// SIMATIC S7-200 SMART project (STEP 7-Micro/WIN SMART), CPU SR40

SYMBOL_TABLE 系统符号
Always_On        SM0.0    // 始终接通
First_Scan_On    SM0.1    // 仅在第一个扫描周期时接通
END_SYMBOL_TABLE

ORGANIZATION_BLOCK MAIN:OB1
TITLE=程序注释
BEGIN
Network 1
// 程序段注释
LD     First_Scan_On:SM0.1   //第一次扫描时
MOVB   16#7, QB0             //设置彩灯的初始状态，最低3位的灯被点亮
ATCH   INT_0:INT0, 21        //指定T32定时时间到时执行中断程序INT_0
ENI                          //允许全局中断
Network 2
LDN    M0.0                  //T32和M0.0组成脉冲发生器
TON    T32, 3000             //T32 的预设值为3000ms
Network 3
LD     T32
=      M0.0
END_ORGANIZATION_BLOCK

INTERRUPT_BLOCK INT_0:INT0
TITLE=中断例程注释
BEGIN
Network 1
// 程序段注释
LD     Always_On:SM0.0
RLB    QB0, 1                //彩灯循环左移1位
END_INTERRUPT_BLOCK
